// TIA Portal V17 export
// export: Created 2023-04-03T06:31:37.4692763Z, ExportSetting WithDefaults, DisplayName Totally Integrated Automation Portal, DisplayVersion V17 Update 4, DisplayName TIA Portal Openness, DisplayVersion V17 Update 4, DisplayName TIA Portal Version Control Interface, DisplayVersion V17, DisplayName STEP 7 Professional, DisplayVersion V17 Update 4, DisplayName STEP 7 Safety, DisplayVersion V17, DisplayName WinCC Professional, DisplayVersion V17 Update 4
ORGANIZATION_BLOCK "Cyclic interrupt 100ms"   // OB33, LAD, CyclicInterrupt
{ S7_Optimized_Access := 'TRUE' }
VERSION : 0.1
// stored: AutoNumber false, IsIECCheckEnabled false, SetENOAutomatically false
   VAR_INPUT
      Initial_Call : Bool;   // Initial call of this OB
      Event_Count : Int;   // Events discarded
   END_VAR
BEGIN

REGION Network 1
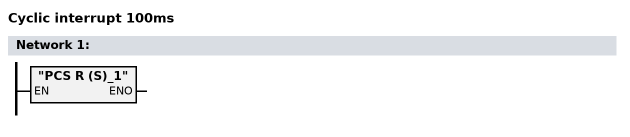
   RUNG wire#powerrail
      "PCS R (S)_1"()
   END_RUNG
   // the same network as SCL:
   "PCS R (S)_1"();
END_REGION
END_ORGANIZATION_BLOCK
